// TIA Portal V19 export
FUNCTION_BLOCK "RollformerLubr_FB"   // FB163, LAD
TITLE = Rollfomer Lubr
// stored: MemoryReserve 100, SetENOAutomatically false
   VAR_INPUT
      AreaInterface : "AreaInterface";
   END_VAR
   VAR_OUTPUT
      MachineInterface : "MachineInterface";
   END_VAR
   VAR
      Pump : "Lubr_Motor";
      Valves1 : "Lubr_Valve";
      Valves2 { S7_SetPoint := 'True'} : "Lubr_Valve";
      Valves3 { S7_SetPoint := 'True'} : "Lubr_Valve";
   END_VAR
BEGIN

REGION Network 2: <<< POMPA PRINCIPALE >>>
END_REGION

REGION Network 3: Data In
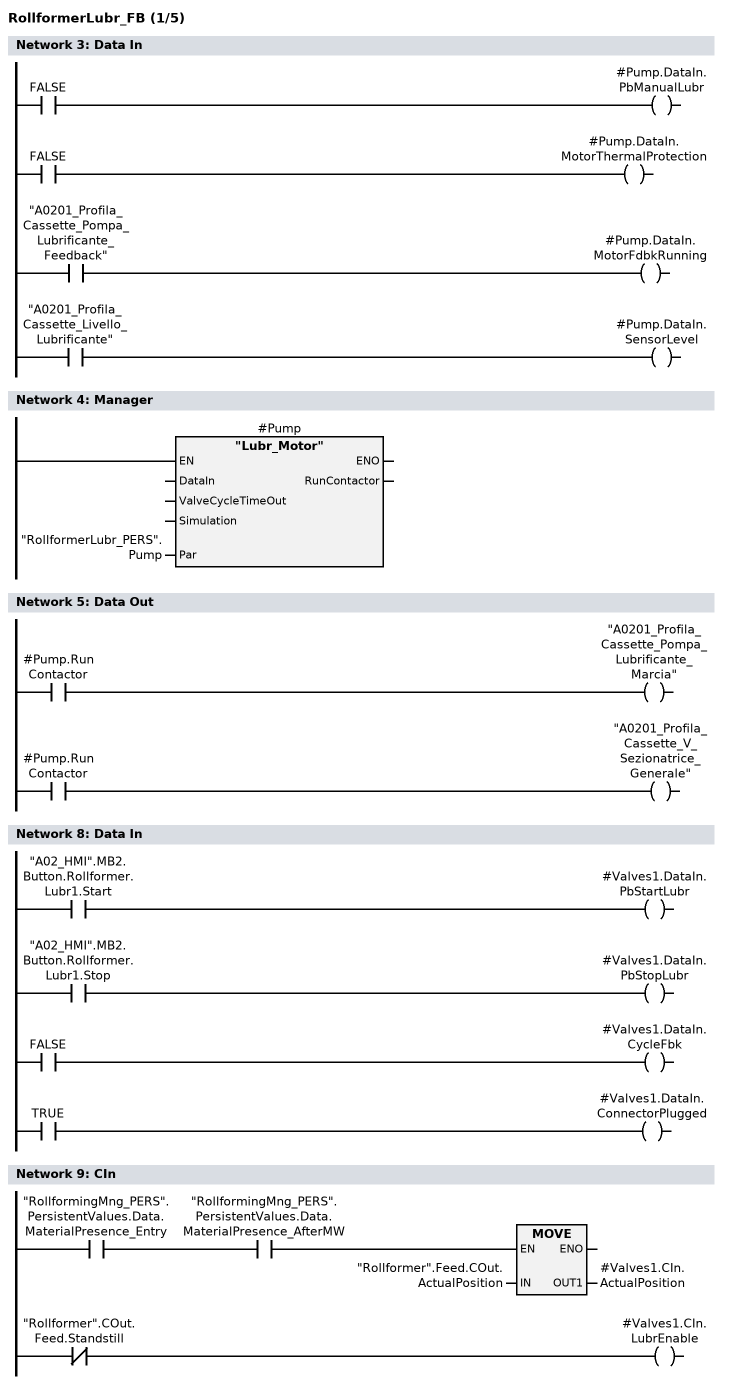
   RUNG wire#powerrail
      Contact( FALSE )
      Coil( #Pump.DataIn.PbManualLubr )
   END_RUNG
   RUNG wire#powerrail
      Contact( FALSE )
      Coil( #Pump.DataIn.MotorThermalProtection )
   END_RUNG
   RUNG wire#powerrail
      Contact( "A0201_Profila_Cassette_Pompa_Lubrificante_Feedback" )
      Coil( #Pump.DataIn.MotorFdbkRunning )
   END_RUNG
   RUNG wire#powerrail
      Contact( "A0201_Profila_Cassette_Livello_Lubrificante" )
      Coil( #Pump.DataIn.SensorLevel )
   END_RUNG
   // the same network as SCL:
   #Pump.DataIn.PbManualLubr := FALSE;
   #Pump.DataIn.MotorThermalProtection := FALSE;
   #Pump.DataIn.MotorFdbkRunning := "A0201_Profila_Cassette_Pompa_Lubrificante_Feedback";
   #Pump.DataIn.SensorLevel := "A0201_Profila_Cassette_Livello_Lubrificante";
END_REGION

REGION Network 4: Manager
   RUNG wire#powerrail
      #Pump(DataIn :=, ValveCycleTimeOut :=, Simulation :=, Par := "RollformerLubr_PERS".Pump, RunContactor =>)
   END_RUNG
   // the same network as SCL:
   #Pump(Par := "RollformerLubr_PERS".Pump);   // "Lubr_Motor"
END_REGION

REGION Network 5: Data Out
   RUNG wire#powerrail
      Contact( #Pump.RunContactor )
      Coil( "A0201_Profila_Cassette_Pompa_Lubrificante_Marcia" )
   END_RUNG
   RUNG wire#powerrail
      Contact( #Pump.RunContactor )
      Coil( "A0201_Profila_Cassette_V_Sezionatrice_Generale" )
   END_RUNG
   // the same network as SCL:
   "A0201_Profila_Cassette_Pompa_Lubrificante_Marcia" := #Pump.RunContactor;
   "A0201_Profila_Cassette_V_Sezionatrice_Generale" := #Pump.RunContactor;
END_REGION

REGION Network 7: <<< CASSETTA 1 VALVOLE >>>
END_REGION

REGION Network 8: Data In
   RUNG wire#powerrail
      Contact( "A02_HMI".MB2.Button.Rollformer.Lubr1.Start )
      Coil( #Valves1.DataIn.PbStartLubr )
   END_RUNG
   RUNG wire#powerrail
      Contact( "A02_HMI".MB2.Button.Rollformer.Lubr1.Stop )
      Coil( #Valves1.DataIn.PbStopLubr )
   END_RUNG
   RUNG wire#powerrail
      Contact( FALSE )
      Coil( #Valves1.DataIn.CycleFbk )
   END_RUNG
   RUNG wire#powerrail
      Contact( TRUE )
      Coil( #Valves1.DataIn.ConnectorPlugged )
   END_RUNG
   // the same network as SCL:
   #Valves1.DataIn.PbStartLubr := "A02_HMI".MB2.Button.Rollformer.Lubr1.Start;
   #Valves1.DataIn.PbStopLubr := "A02_HMI".MB2.Button.Rollformer.Lubr1.Stop;
   #Valves1.DataIn.CycleFbk := FALSE;
   #Valves1.DataIn.ConnectorPlugged := TRUE;
END_REGION

REGION Network 9: CIn
   RUNG wire#powerrail
      Contact( "RollformingMng_PERS".PersistentValues.Data.MaterialPresence_Entry )
      Contact( "RollformingMng_PERS".PersistentValues.Data.MaterialPresence_AfterMW )
      Move(in := "Rollformer".Feed.COut.ActualPosition, out1 => #Valves1.CIn.ActualPosition)
   END_RUNG
   RUNG wire#powerrail
      I_Contact( "Rollformer".COut.Feed.Standstill )
      Coil( #Valves1.CIn.LubrEnable )
   END_RUNG
   // the same network as SCL:
   IF "RollformingMng_PERS".PersistentValues.Data.MaterialPresence_Entry AND "RollformingMng_PERS".PersistentValues.Data.MaterialPresence_AfterMW THEN
       #Valves1.CIn.ActualPosition := "Rollformer".Feed.COut.ActualPosition;
   END_IF;
   #Valves1.CIn.LubrEnable := NOT "Rollformer".COut.Feed.Standstill;
END_REGION

REGION Network 10: Manager
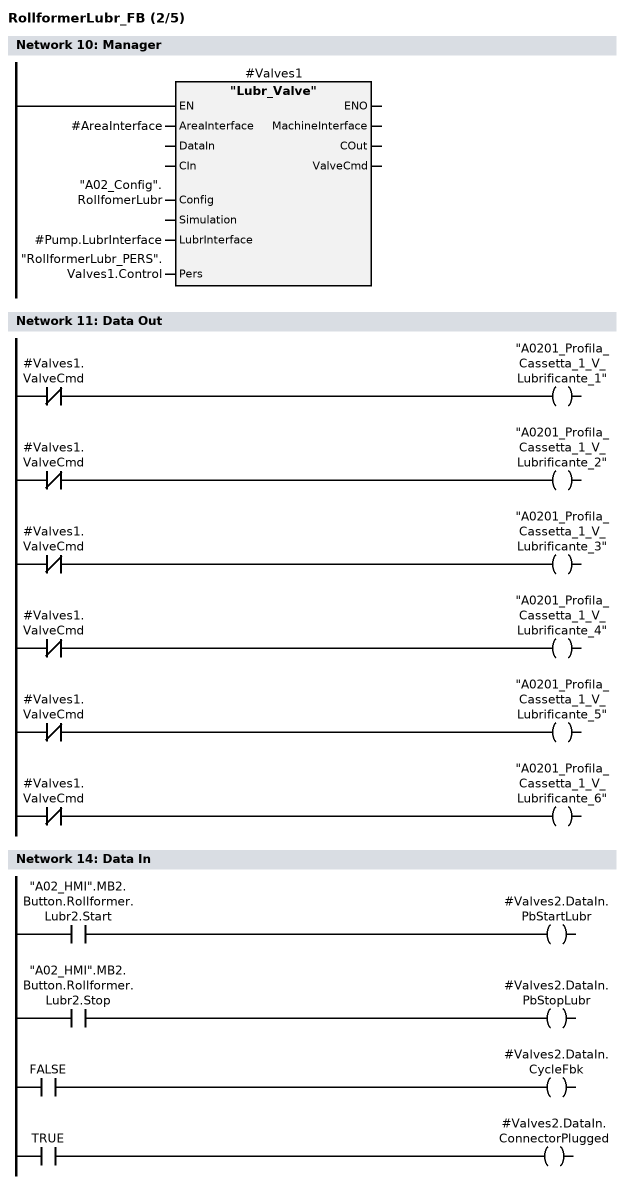
   RUNG wire#powerrail
      #Valves1(AreaInterface := #AreaInterface, DataIn :=, CIn :=, Config := "A02_Config".RollfomerLubr, Simulation :=, LubrInterface := #Pump.LubrInterface, Pers := "RollformerLubr_PERS".Valves1.Control, MachineInterface =>, COut =>, ValveCmd =>)
   END_RUNG
   // the same network as SCL:
   #Valves1(AreaInterface := #AreaInterface,   // "Lubr_Valve"
            Config := "A02_Config".RollfomerLubr,
            LubrInterface := #Pump.LubrInterface,
            Pers := "RollformerLubr_PERS".Valves1.Control);
END_REGION

REGION Network 11: Data Out
   RUNG wire#powerrail
      I_Contact( #Valves1.ValveCmd )
      Coil( "A0201_Profila_Cassetta_1_V_Lubrificante_1" )
   END_RUNG
   RUNG wire#powerrail
      I_Contact( #Valves1.ValveCmd )
      Coil( "A0201_Profila_Cassetta_1_V_Lubrificante_2" )
   END_RUNG
   RUNG wire#powerrail
      I_Contact( #Valves1.ValveCmd )
      Coil( "A0201_Profila_Cassetta_1_V_Lubrificante_3" )
   END_RUNG
   RUNG wire#powerrail
      I_Contact( #Valves1.ValveCmd )
      Coil( "A0201_Profila_Cassetta_1_V_Lubrificante_4" )
   END_RUNG
   RUNG wire#powerrail
      I_Contact( #Valves1.ValveCmd )
      Coil( "A0201_Profila_Cassetta_1_V_Lubrificante_5" )
   END_RUNG
   RUNG wire#powerrail
      I_Contact( #Valves1.ValveCmd )
      Coil( "A0201_Profila_Cassetta_1_V_Lubrificante_6" )
   END_RUNG
   // the same network as SCL:
   "A0201_Profila_Cassetta_1_V_Lubrificante_1" := NOT #Valves1.ValveCmd;
   "A0201_Profila_Cassetta_1_V_Lubrificante_2" := NOT #Valves1.ValveCmd;
   "A0201_Profila_Cassetta_1_V_Lubrificante_3" := NOT #Valves1.ValveCmd;
   "A0201_Profila_Cassetta_1_V_Lubrificante_4" := NOT #Valves1.ValveCmd;
   "A0201_Profila_Cassetta_1_V_Lubrificante_5" := NOT #Valves1.ValveCmd;
   "A0201_Profila_Cassetta_1_V_Lubrificante_6" := NOT #Valves1.ValveCmd;
END_REGION

REGION Network 13: <<< CASSETTA 2 VALVOLE >>>
END_REGION

REGION Network 14: Data In
   RUNG wire#powerrail
      Contact( "A02_HMI".MB2.Button.Rollformer.Lubr2.Start )
      Coil( #Valves2.DataIn.PbStartLubr )
   END_RUNG
   RUNG wire#powerrail
      Contact( "A02_HMI".MB2.Button.Rollformer.Lubr2.Stop )
      Coil( #Valves2.DataIn.PbStopLubr )
   END_RUNG
   RUNG wire#powerrail
      Contact( FALSE )
      Coil( #Valves2.DataIn.CycleFbk )
   END_RUNG
   RUNG wire#powerrail
      Contact( TRUE )
      Coil( #Valves2.DataIn.ConnectorPlugged )
   END_RUNG
   // the same network as SCL:
   #Valves2.DataIn.PbStartLubr := "A02_HMI".MB2.Button.Rollformer.Lubr2.Start;
   #Valves2.DataIn.PbStopLubr := "A02_HMI".MB2.Button.Rollformer.Lubr2.Stop;
   #Valves2.DataIn.CycleFbk := FALSE;
   #Valves2.DataIn.ConnectorPlugged := TRUE;
END_REGION

REGION Network 15: CIn
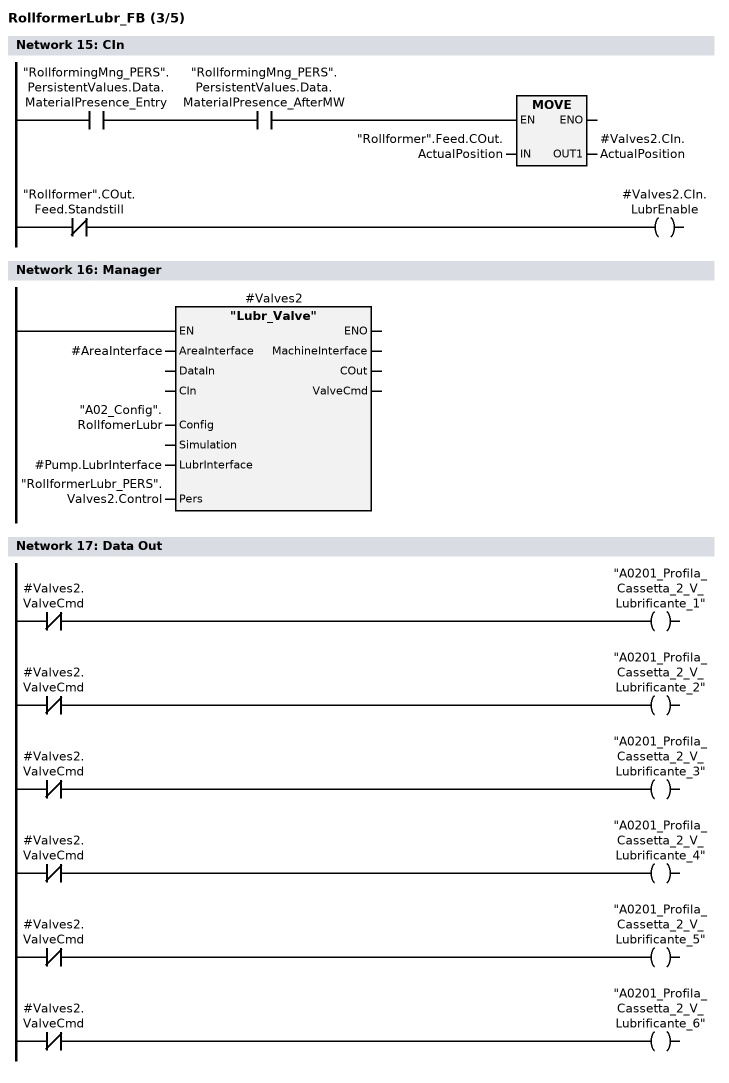
   RUNG wire#powerrail
      Contact( "RollformingMng_PERS".PersistentValues.Data.MaterialPresence_Entry )
      Contact( "RollformingMng_PERS".PersistentValues.Data.MaterialPresence_AfterMW )
      Move(in := "Rollformer".Feed.COut.ActualPosition, out1 => #Valves2.CIn.ActualPosition)
   END_RUNG
   RUNG wire#powerrail
      I_Contact( "Rollformer".COut.Feed.Standstill )
      Coil( #Valves2.CIn.LubrEnable )
   END_RUNG
   // the same network as SCL:
   IF "RollformingMng_PERS".PersistentValues.Data.MaterialPresence_Entry AND "RollformingMng_PERS".PersistentValues.Data.MaterialPresence_AfterMW THEN
       #Valves2.CIn.ActualPosition := "Rollformer".Feed.COut.ActualPosition;
   END_IF;
   #Valves2.CIn.LubrEnable := NOT "Rollformer".COut.Feed.Standstill;
END_REGION

REGION Network 16: Manager
   RUNG wire#powerrail
      #Valves2(AreaInterface := #AreaInterface, DataIn :=, CIn :=, Config := "A02_Config".RollfomerLubr, Simulation :=, LubrInterface := #Pump.LubrInterface, Pers := "RollformerLubr_PERS".Valves2.Control, MachineInterface =>, COut =>, ValveCmd =>)
   END_RUNG
   // the same network as SCL:
   #Valves2(AreaInterface := #AreaInterface,   // "Lubr_Valve"
            Config := "A02_Config".RollfomerLubr,
            LubrInterface := #Pump.LubrInterface,
            Pers := "RollformerLubr_PERS".Valves2.Control);
END_REGION

REGION Network 17: Data Out
   RUNG wire#powerrail
      I_Contact( #Valves2.ValveCmd )
      Coil( "A0201_Profila_Cassetta_2_V_Lubrificante_1" )
   END_RUNG
   RUNG wire#powerrail
      I_Contact( #Valves2.ValveCmd )
      Coil( "A0201_Profila_Cassetta_2_V_Lubrificante_2" )
   END_RUNG
   RUNG wire#powerrail
      I_Contact( #Valves2.ValveCmd )
      Coil( "A0201_Profila_Cassetta_2_V_Lubrificante_3" )
   END_RUNG
   RUNG wire#powerrail
      I_Contact( #Valves2.ValveCmd )
      Coil( "A0201_Profila_Cassetta_2_V_Lubrificante_4" )
   END_RUNG
   RUNG wire#powerrail
      I_Contact( #Valves2.ValveCmd )
      Coil( "A0201_Profila_Cassetta_2_V_Lubrificante_5" )
   END_RUNG
   RUNG wire#powerrail
      I_Contact( #Valves2.ValveCmd )
      Coil( "A0201_Profila_Cassetta_2_V_Lubrificante_6" )
   END_RUNG
   // the same network as SCL:
   "A0201_Profila_Cassetta_2_V_Lubrificante_1" := NOT #Valves2.ValveCmd;
   "A0201_Profila_Cassetta_2_V_Lubrificante_2" := NOT #Valves2.ValveCmd;
   "A0201_Profila_Cassetta_2_V_Lubrificante_3" := NOT #Valves2.ValveCmd;
   "A0201_Profila_Cassetta_2_V_Lubrificante_4" := NOT #Valves2.ValveCmd;
   "A0201_Profila_Cassetta_2_V_Lubrificante_5" := NOT #Valves2.ValveCmd;
   "A0201_Profila_Cassetta_2_V_Lubrificante_6" := NOT #Valves2.ValveCmd;
END_REGION

REGION Network 19: <<< CASSETTA 3 VALVOLE >>>
END_REGION

REGION Network 20: Data In
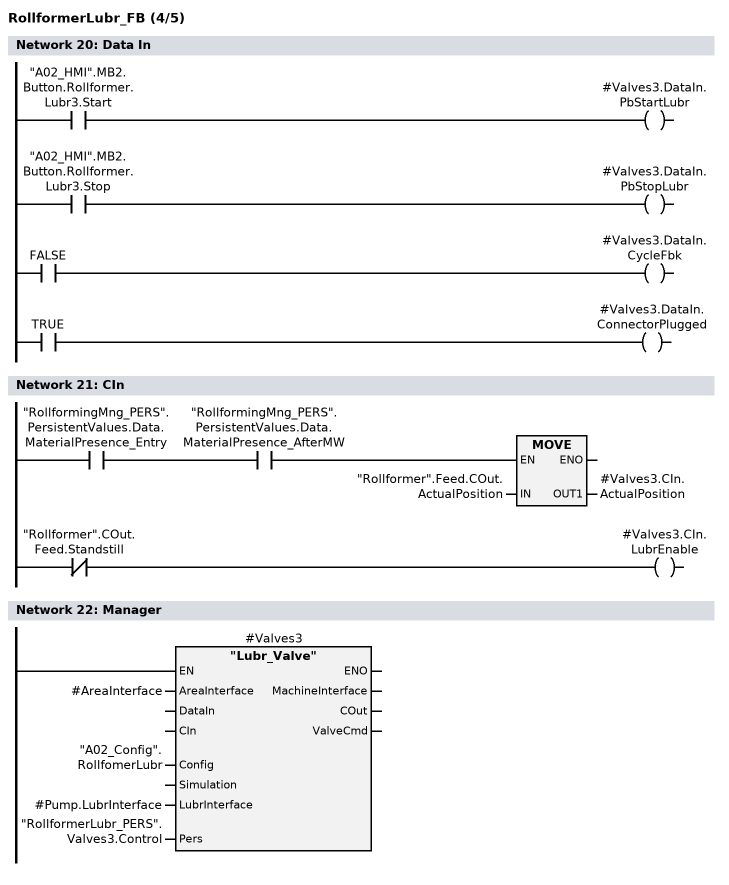
   RUNG wire#powerrail
      Contact( "A02_HMI".MB2.Button.Rollformer.Lubr3.Start )
      Coil( #Valves3.DataIn.PbStartLubr )
   END_RUNG
   RUNG wire#powerrail
      Contact( "A02_HMI".MB2.Button.Rollformer.Lubr3.Stop )
      Coil( #Valves3.DataIn.PbStopLubr )
   END_RUNG
   RUNG wire#powerrail
      Contact( FALSE )
      Coil( #Valves3.DataIn.CycleFbk )
   END_RUNG
   RUNG wire#powerrail
      Contact( TRUE )
      Coil( #Valves3.DataIn.ConnectorPlugged )
   END_RUNG
   // the same network as SCL:
   #Valves3.DataIn.PbStartLubr := "A02_HMI".MB2.Button.Rollformer.Lubr3.Start;
   #Valves3.DataIn.PbStopLubr := "A02_HMI".MB2.Button.Rollformer.Lubr3.Stop;
   #Valves3.DataIn.CycleFbk := FALSE;
   #Valves3.DataIn.ConnectorPlugged := TRUE;
END_REGION

REGION Network 21: CIn
   RUNG wire#powerrail
      Contact( "RollformingMng_PERS".PersistentValues.Data.MaterialPresence_Entry )
      Contact( "RollformingMng_PERS".PersistentValues.Data.MaterialPresence_AfterMW )
      Move(in := "Rollformer".Feed.COut.ActualPosition, out1 => #Valves3.CIn.ActualPosition)
   END_RUNG
   RUNG wire#powerrail
      I_Contact( "Rollformer".COut.Feed.Standstill )
      Coil( #Valves3.CIn.LubrEnable )
   END_RUNG
   // the same network as SCL:
   IF "RollformingMng_PERS".PersistentValues.Data.MaterialPresence_Entry AND "RollformingMng_PERS".PersistentValues.Data.MaterialPresence_AfterMW THEN
       #Valves3.CIn.ActualPosition := "Rollformer".Feed.COut.ActualPosition;
   END_IF;
   #Valves3.CIn.LubrEnable := NOT "Rollformer".COut.Feed.Standstill;
END_REGION

REGION Network 22: Manager
   RUNG wire#powerrail
      #Valves3(AreaInterface := #AreaInterface, DataIn :=, CIn :=, Config := "A02_Config".RollfomerLubr, Simulation :=, LubrInterface := #Pump.LubrInterface, Pers := "RollformerLubr_PERS".Valves3.Control, MachineInterface =>, COut =>, ValveCmd =>)
   END_RUNG
   // the same network as SCL:
   #Valves3(AreaInterface := #AreaInterface,   // "Lubr_Valve"
            Config := "A02_Config".RollfomerLubr,
            LubrInterface := #Pump.LubrInterface,
            Pers := "RollformerLubr_PERS".Valves3.Control);
END_REGION

REGION Network 23: Data Out
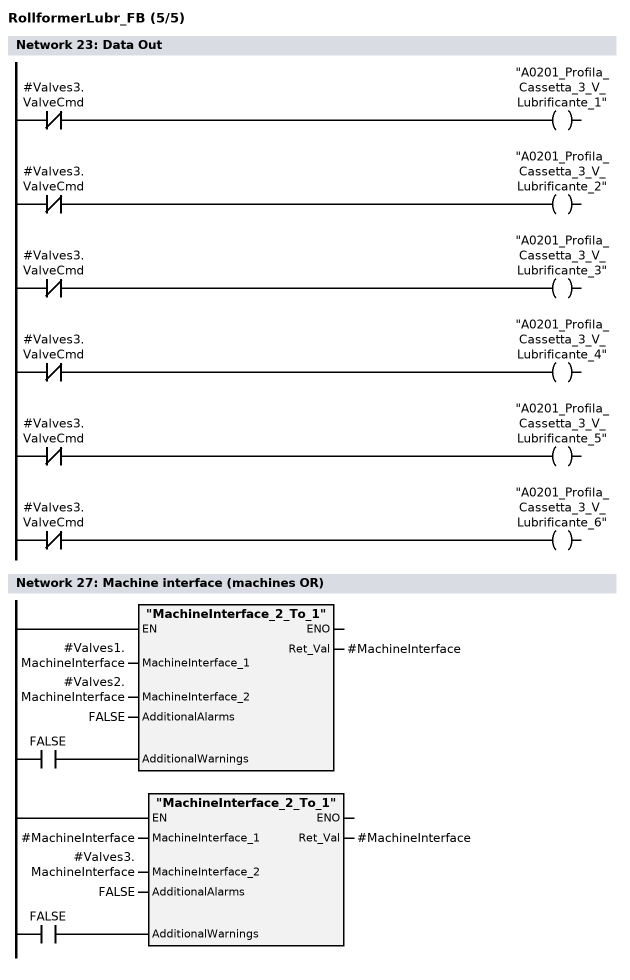
   RUNG wire#powerrail
      I_Contact( #Valves3.ValveCmd )
      Coil( "A0201_Profila_Cassetta_3_V_Lubrificante_1" )
   END_RUNG
   RUNG wire#powerrail
      I_Contact( #Valves3.ValveCmd )
      Coil( "A0201_Profila_Cassetta_3_V_Lubrificante_2" )
   END_RUNG
   RUNG wire#powerrail
      I_Contact( #Valves3.ValveCmd )
      Coil( "A0201_Profila_Cassetta_3_V_Lubrificante_3" )
   END_RUNG
   RUNG wire#powerrail
      I_Contact( #Valves3.ValveCmd )
      Coil( "A0201_Profila_Cassetta_3_V_Lubrificante_4" )
   END_RUNG
   RUNG wire#powerrail
      I_Contact( #Valves3.ValveCmd )
      Coil( "A0201_Profila_Cassetta_3_V_Lubrificante_5" )
   END_RUNG
   RUNG wire#powerrail
      I_Contact( #Valves3.ValveCmd )
      Coil( "A0201_Profila_Cassetta_3_V_Lubrificante_6" )
   END_RUNG
   // the same network as SCL:
   "A0201_Profila_Cassetta_3_V_Lubrificante_1" := NOT #Valves3.ValveCmd;
   "A0201_Profila_Cassetta_3_V_Lubrificante_2" := NOT #Valves3.ValveCmd;
   "A0201_Profila_Cassetta_3_V_Lubrificante_3" := NOT #Valves3.ValveCmd;
   "A0201_Profila_Cassetta_3_V_Lubrificante_4" := NOT #Valves3.ValveCmd;
   "A0201_Profila_Cassetta_3_V_Lubrificante_5" := NOT #Valves3.ValveCmd;
   "A0201_Profila_Cassetta_3_V_Lubrificante_6" := NOT #Valves3.ValveCmd;
END_REGION

REGION Network 24: Data Out
END_REGION

REGION Network 27: Machine interface (machines OR)
   RUNG wire#powerrail
      "MachineInterface_2_To_1"(AdditionalWarnings := wire#w1, MachineInterface_1 := #Valves1.MachineInterface, MachineInterface_2 := #Valves2.MachineInterface, AdditionalAlarms := FALSE, Ret_Val => #MachineInterface)
   END_RUNG
   RUNG wire#powerrail
      Contact( FALSE )
   END_RUNG wire#w1
   RUNG wire#powerrail
      "MachineInterface_2_To_1"(AdditionalWarnings := wire#w2, MachineInterface_1 := #MachineInterface, MachineInterface_2 := #Valves3.MachineInterface, AdditionalAlarms := FALSE, Ret_Val => #MachineInterface)
   END_RUNG
   RUNG wire#powerrail
      Contact( FALSE )
   END_RUNG wire#w2
   // the same network as SCL:
   #MachineInterface := "MachineInterface_2_To_1"(MachineInterface_1 := #Valves1.MachineInterface,
                           MachineInterface_2 := #Valves2.MachineInterface,
                           AdditionalAlarms := FALSE,
                           AdditionalWarnings := FALSE);
   #MachineInterface := "MachineInterface_2_To_1"(MachineInterface_1 := #MachineInterface,
                           MachineInterface_2 := #Valves3.MachineInterface,
                           AdditionalAlarms := FALSE,
                           AdditionalWarnings := FALSE);
END_REGION
END_FUNCTION_BLOCK
